// TIA Portal project "Project1" (V20)

(* hardware
DEVICE "S7-1200 station_1"  S7-1200 Station
   slot 0: "Rack_0"  S7-1200 Rack  Rack  V1.0
   slot 1: "PLC_1"  CPU 1215C DC/DC/Rly  6ES7 215-1HG40-0XB0  V4.6
DEVICE "HMI_1"  KTP700 Basic PN Portrait
   slot 0: "HMI_1"  KTP700 Basic PN Portrait  6AV2 123-2GB03-0AX0  17.0.0.0
   slot 1: "HMI_RT_1"  KTP700 Basic PN Portrait  6AV2 123-2GB03-0AX0  17.0.0.0
   slot 5: "HMI_1.IE_CP_1"  PROFINET Interface  17.0.0.0
      slot 1: "PROFINET Interface_1"  PROFINET Interface
         slot 1: "Port_1"  Port
*)

// ===== PLC "PLC_1"  CPU 1215C DC/DC/Rly =====

VAR_GLOBAL   // PLC tag table "Default tag table"
   "Start" AT %M0.0 : Bool;
   "Motor" AT %M1.0 : Bool;
   "Stop Push buttom" AT %M0.1 : Bool;
   "Stop my model" AT %M1.1 : Bool;
   "Blue Bt" AT %M0.4 : Bool;
   "set" AT %M0.3 : Bool;
   "reset" AT %M0.5 : Bool;
   "t1_sig" AT %M0.2 : Bool;
   "t2_sig" AT %M0.6 : Bool;
   "e-time" AT %MD2 : Time;
   "count_sig" AT %M0.7 : Bool;
   "light" AT %M1.2 : Bool;
END_VAR

// folder: System blocks/Program resources

DATA_BLOCK "IEC_Counter_0_DB"   // DB1
{ S7_Optimized_Access := 'TRUE' }
AUTHOR : Simatic
FAMILY : IEC
NAME : CNTR
VERSION : 1.0
// stored: InstanceOfName IEC_COUNTER
"IEC_COUNTER"
BEGIN
END_DATA_BLOCK

DATA_BLOCK "IEC_Timer_0_DB"   // DB3
{ S7_Optimized_Access := 'TRUE' }
AUTHOR : Simatic
FAMILY : IEC
NAME : IEC_TMR
VERSION : 1.0
// stored: InstanceOfName IEC_TIMER
"IEC_TIMER"
BEGIN
END_DATA_BLOCK

DATA_BLOCK "IEC_Timer_0_DB_1"   // DB4
{ S7_Optimized_Access := 'TRUE' }
AUTHOR : Simatic
FAMILY : IEC
NAME : IEC_TMR
VERSION : 1.0
// stored: InstanceOfName IEC_TIMER
"IEC_TIMER"
BEGIN
END_DATA_BLOCK

// folder: (top level)

ORGANIZATION_BLOCK "Main"   // OB1, LAD, ProgramCycle
TITLE = "Main Program Sweep (Cycle)"
{ S7_Optimized_Access := 'TRUE' }
VERSION : 0.1
   VAR_INPUT
      Initial_Call : Bool;   // Initial call of this OB
      Remanence : Bool;   // =True, if remanent data are available
   END_VAR
   VAR_TEMP
      e_time_2 : Time;
      count : Int;
   END_VAR
BEGIN

REGION Network 1
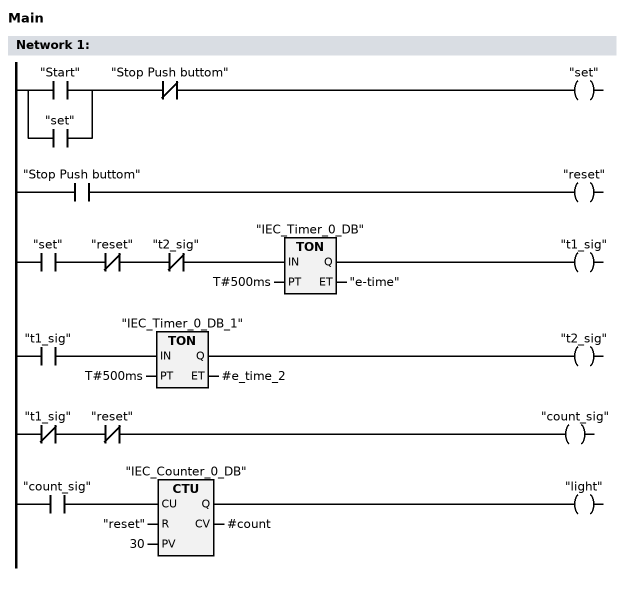
   "set" := ("Start" OR "set") AND NOT "Stop Push buttom";
   "reset" := "Stop Push buttom";
   "IEC_Timer_0_DB".TON(IN := "set" AND NOT "reset" AND NOT "t2_sig", PT := T#500ms, ET => "e-time");
   "t1_sig" := "IEC_Timer_0_DB".Q;
   "IEC_Timer_0_DB_1".TON(IN := "t1_sig", PT := T#500ms, ET => #e_time_2);
   "t2_sig" := "IEC_Timer_0_DB_1".Q;
   "count_sig" := NOT "t1_sig" AND NOT "reset";
   "IEC_Counter_0_DB".CTU(CU := "count_sig", R := "reset", PV := 30, CV => #count);
   "light" := "IEC_Counter_0_DB".Q;
END_REGION
END_ORGANIZATION_BLOCK

(* ===== HMI "HMI_RT_1" =====
system functions are stored by id; their names below are inferred from use
connection "HMI_Connection_1": ETHERNET, SMART_S7_1200_OMS

HMI tags "Default tag table"
   "Tag_ScreenNumber" : UInt, internal
   "StartHMI" : Bool = PLC Start AT %M0.0, 1 s
   "StopHMI" : Bool = PLC "Stop Push buttom" AT %M0.1, 1 s
   "Emergency" : Bool = PLC "Emergency switch" AT %M0.2, 1 s
   "MotorH" : Bool = PLC Motor AT %M1.0, 1 s
   "StopMyModel" : Bool = PLC "Stop my model" AT %M1.1, 1 s
   "YellowLED" : Bool = PLC "Yellow LED" AT %Q0.2, 1 s
   "Blue" : Bool = PLC "Blue Bt" AT %M0.4, 1 s

Template "Template_1" 480x800
   Button "Start screen" at 428,61 size 50x71; TextOff 'Start screen'; PictureOff "NavigateHome_KTP700_Basic_PN_Portrait_TR"; PictureOn "NavigateHome_KTP700_Basic_PN_Portrait_TR"
      on Release: ActivateScreen("Root screen", 0)
   Button "Alarms" at 428,172 size 50x71; TextOff 'Alarms'; PictureOff "AlarmDisplay_KTP700_Basic_PN_Portrait_TR"; PictureOn "AlarmDisplay_KTP700_Basic_PN_Portrait_TR"
      on Release: function_ef3f5d25("Alarm window_Unacknowledged", -1)
   Button "Template_Button" at 428,283 size 50x71; TextOff 'Text'
   Button "Template_Button_1" at 428,394 size 50x71; TextOff 'Text'
   Button "Template_Button_2" at 428,505 size 50x71; TextOff 'Text'
   Button "Template_Button_3" at 428,616 size 50x71; TextOff 'Text'
   Button "Exit" at 428,727 size 50x71; TextOff 'Exit'; PictureOff "ExitRuntime_KTP700_Basic_PN_Portrait_TR"; PictureOn "ExitRuntime_KTP700_Basic_PN_Portrait_TR"
      on Release: StopRuntime(0)
   SymbolicIOField "Symbolic_IO_Field_Screen" at 109,11 size 264x38; TextOff '0'; TextOn '1'; TextList "TextList_ScreenNames"
      ProcessValue <- "Tag_ScreenNumber"
      on Change: ActivateScreenByNumber("Tag_ScreenNumber", 0)
   DateTimeField "HmiScreenItemData" at 375,30 size 105x30
   DateTimeField "HmiScreenItemData_1" at 375,0 size 105x30
   GraphicView "Logo" at 0,0 size 107x60; Picture "Logo of HMI_1"

screen "Root screen" 480x800, template "Template_1"
   on GenerateScreen: SetTag("Tag_ScreenNumber", 1)
   TextField "HmiScreenItemData" at 43,404 size 343x46; Text 'Welcome to HMI_1 (KTP700 Basic+ PN Portrait)!'
*)